{attribute 'linkalways'} 
{attribute 'no_explicit_call' := 'This FB is a CLASS and must be accessed using methods or properties'}
{attribute 'enable_dynamic_creation'}
FUNCTION_BLOCK Node_F_VN_ReadDataMatrixCode EXTENDS VisionNode
VAR
    ipSrcImage : _ITcVnImage;
    ipDecodedData : _ITcVnContainer;
    hrPrev : _HRESULT(S_OK);
	hresult : _HRESULT(S_OK);
END_VAR

METHOD PUBLIC  Clone : I_Node
VAR
	pNode : POINTER TO Node_F_VN_ReadDataMatrixCode;
END_VAR
pNode := __NEW(Node_F_VN_ReadDataMatrixCode);
Clone := pNode^;
END_METHOD

METHOD FB_init : BOOL
VAR_INPUT
	bInitRetains : BOOL; // if TRUE, the retain variables are initialized (warm start / cold start)
	bInCopyCode : BOOL;  // if TRUE, the instance afterwards gets moved into the copy code (online change)
END_VAR
AddInput('ipSrcImage', ipSrcImage);
AddInput('hrPrev', hrPrev);
AddOutput('ipDecodedData', ipDecodedData);
AddOutput('hresult',hresult);
END_METHOD

METHOD PROTECTED OnExecute : HRESULT
hresult.Value := F_VN_ReadDataMatrixCode(
	ipSrcImage := ipSrcImage.Value,
    ipDecodedData := ipDecodedData.Value,
	hrPrev:= hrPrev.Value);
END_METHOD

METHOD PUBLIC PreExecutionCheck
VAR_INPUT
	Check : I_PreExecutionChecks;
END_VAR
Check.IsTrue(ipSrcImage.IsValid, 'ipSrcImage must contain an image');
Check.IsTrue((ipSrcImage.HasChannelCount(1) OR ipSrcImage.HasChannelCount(3)), 'ipSrcImage must have 1 channel');
Check.IsTrue(ipSrcImage.IsPixelDepth(8), 'ipSrcImage must have 8 bit pixel depth');
END_METHOD

END_FUNCTION_BLOCK

(* stored: Version 1.1.0.1, ProductVersion 3.1.4024.13
   POU Node_F_VN_ReadDataMatrixCode: Id {48758f93-2f36-0f89-177c-e2ea6a44e294}, SpecialFunc None
   Folder Constructor: Id {e164ae47-9b7c-01c6-285a-e6d05e9762f7}
   Method Clone: Id {89399bb7-69a4-096c-1548-89824b3e7914}
   Method FB_init: Id {7055f3ac-550b-0685-17b2-5ec52a3ec544}
   Method OnExecute: Id {e2f83839-48f4-0c14-279f-5561be136c3b}
   Method PreExecutionCheck: Id {1bb05a25-6444-0410-22bb-387924db59f7} *)
